// SIMATIC S7-200 project (STEP 7-Micro/WIN), CPU 221 REL 01.10

SYMBOL_TABLE USUARIO1
PM               I0.0     // Pulsador de marcha
PG               I0.1     // Pulsador de paro (NC)
FC               I0.2     // Final de carrera detección paquete
a0               I0.3     // Captador magnético actuador A contraído
a1               I0.4     // Captador magnético actuador A expandido
b0               I0.5     // Captador magnético actuador B contraído
b1               I0.6     // Captador magnético actuador B expandido
A_POS            Q0.0     // Expandir actuador A
A_NEG            Q0.1     // Contraer actuador A
B_POS            Q0.2     // Expandir actuador B
B_NEG            Q0.3     // Contraer actuador B
C                Q0.4     // Activar salida de cajas
END_SYMBOL_TABLE

ORGANIZATION_BLOCK PRINCIPAL:OB1
TITLE=COMENTARIOS DEL PROGRAMA
BEGIN
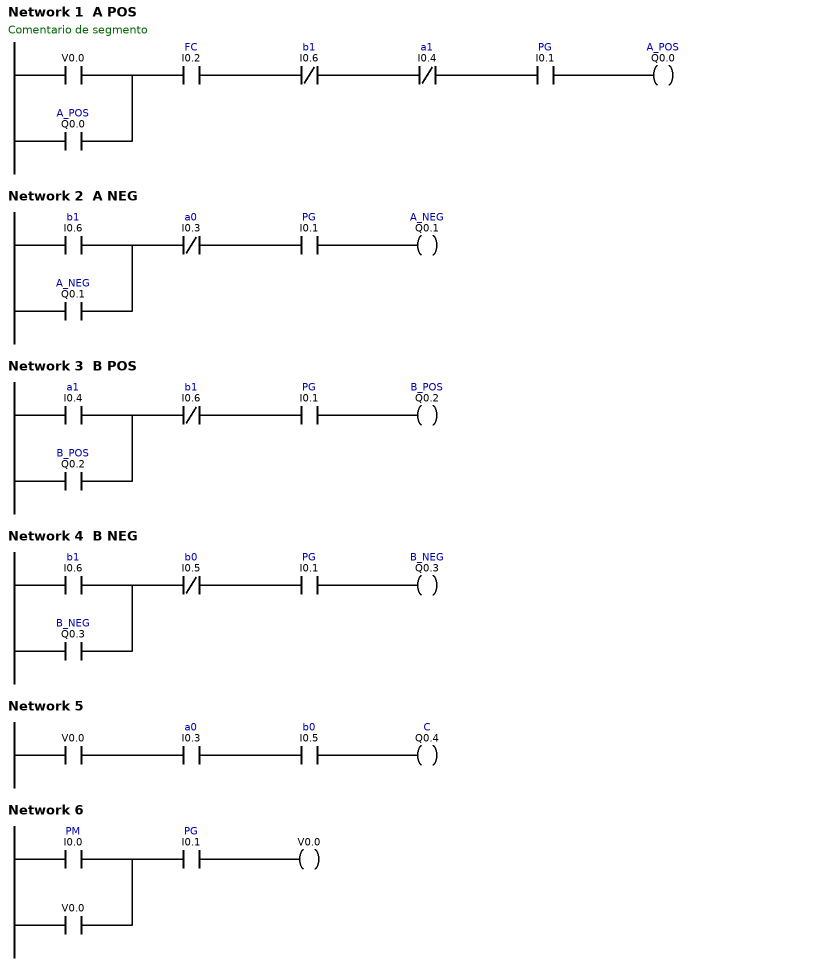
Network 1 // A POS
// Comentario de segmento
LD     V0.0
O      A_POS:Q0.0
A      FC:I0.2
AN     b1:I0.6
AN     a1:I0.4
A      PG:I0.1
=      A_POS:Q0.0
Network 2 // A NEG
LD     b1:I0.6
O      A_NEG:Q0.1
AN     a0:I0.3
A      PG:I0.1
=      A_NEG:Q0.1
Network 3 // B POS

LD     a1:I0.4
O      B_POS:Q0.2
AN     b1:I0.6
A      PG:I0.1
=      B_POS:Q0.2
Network 4 // B NEG
LD     b1:I0.6
O      B_NEG:Q0.3
AN     b0:I0.5
A      PG:I0.1
=      B_NEG:Q0.3
Network 5
LD     V0.0
A      a0:I0.3
A      b0:I0.5
=      C:Q0.4
Network 6
LD     PM:I0.0
O      V0.0
A      PG:I0.1
=      V0.0
END_ORGANIZATION_BLOCK
